{attribute 'GeneratedUsingTerminal: EL4024-0000-0016'}
{attribute addProperty BoxType "EL4024-0000-0016"}
{attribute addProperty Id "EtcSlaveTerminalBaseAO_Outputs_Channel_1AT %Q*AO_Outputs_Channel_BA7EBB7C2AO_Outputs_Channel_2AT %Q*AO_Outputs_Channel_BA7EBB7C2AO_Outputs_Channel_3AT %Q*AO_Outputs_Channel_BA7EBB7C2AO_Outputs_Channel_4AT %Q*AO_Outputs_Channel_BA7EBB7C2WcStateAT %I*WcState_0B2B16F91InfoDataAT %I*InfoData_32EB74EA10"}
{attribute addProperty CRC "4142960146"}
{attribute addProperty Size "19"}
TYPE EL4024_F6F08E12 EXTENDS EtcSlaveTerminalBase :
STRUCT
	{attribute addProperty Name "AO_Outputs_Channel_1"}
	AO_Outputs_Channel_1 : AO_Outputs_Channel_BA7EBB7C;
	{attribute addProperty Name "AO_Outputs_Channel_2"}
	AO_Outputs_Channel_2 : AO_Outputs_Channel_BA7EBB7C;
	{attribute addProperty Name "AO_Outputs_Channel_3"}
	AO_Outputs_Channel_3 : AO_Outputs_Channel_BA7EBB7C;
	{attribute addProperty Name "AO_Outputs_Channel_4"}
	AO_Outputs_Channel_4 : AO_Outputs_Channel_BA7EBB7C;
	{attribute addProperty Name "WcState"}
	WcState : WcState_0B2B16F9;
	{attribute addProperty Name "InfoData"}
	InfoData : InfoData_32EB74EA;
END_STRUCT
END_TYPE

(* stored: Version 1.2.0.0, ProductVersion 3.1.4024.9
   DUT EL4024_F6F08E12: Id {cdea9114-3acd-4a31-8e81-8c0ed2f7f4bc} *)
